TYPE Color:
    (red, yellow, blue);
END_TYPE

(* stored: ProductVersion 3.1.0.18, Version 1.1.0.1 *)
